// Mitsubishi GX Works2 project: PLC_GROUP_22   PLC: FX3G

// global labels: Global1
VAR_GLOBAL
  StartDayButton AT X007 : BOOL;  (* Switching it starts the work day *)
  ActiveDayLamp AT Y007 : BOOL;  (* A light that is on as long as the work day isn't over *)
  RaspberryRegister AT D1100 : REAL;  (* Raspberry inventory tracker *)
  LemonRegister AT D1102 : REAL;  (* Lemon inventory tracker *)
  PreservativeRegister AT D1104 : REAL;  (* Preservative inventory tracker *)
  GummyRegister AT D1106 : REAL;  (* Gummy inventory tracker *)
  SpecialToggle AT M0 : BOOL;  (* When Toggled - use special recpie values *)
  AnalogInput1 AT D8280 : INT;  (* Inputs a number between 1 to 10 to determine which type of popsicle to manufacture *)
  SaveAnalogInput AT D1108 : REAL;  (* Saves the value of toggled input, connects to a Onctroller to determine M0 *)
  EmergencySwitch AT X005 : BOOL;  (* Emergency break *)
  EmergencyFlag AT M2 : BOOL;  (* Signals to break the program *)
  RasperrySpecialRequirement AT E385.0 : REAL;  (* Raspberry Special requirement *)
  PreservativeSpecialRequirement AT E210.0 : REAL;  (* Preservative special recipe requirement *)
  GummySpecialRequirement AT E70.0 : REAL;  (* Gummy special recipe requirement *)
  RasperryRequirement AT E280.0 : REAL;  (* Rasperry regular recipe requirement *)
  LemonRequirement AT E455.0 : REAL;  (* Lemon regular recipe Requirement *)
  PreservativeRequirement AT E105.0 : REAL;  (* Preservative regular recipe requirement *)
  GummyRequirement AT E28.0 : REAL;  (* Gummy regular recipe requirement *)
  IceCreamStartSwitch AT X001 : BOOL;  (* When toggled - start making ice cream *)
  IceCreamMakingTimer AT TC0 : BOOL;  (* Signals if the ice cream making timer finished *)
  Constant50 AT K050 : INT;  (* The it takes to mix the ice cream *)
  IceCreamLamp AT Y000 : BOOL;  (* Signals Ice cream making in process *)
  IceCreamCompletionTimer AT TS0 : BOOL;  (* Signals the system ice cream completion *)
  CoolingSwitch AT X002 : BOOL;  (* Switch starting the cooling process *)
  IceCreamCompletionFlag AT M4 : BOOL;  (* Signals the system's ice cream completion *)
  CoolingFinishFlag AT M5 : BOOL;  (* Flag signaling the ice cream cooling ended *)
  MixingContainer AT D1110 : REAL;  (* The tank where ice cream and gummy are mixed in *)
  MixTimer AT TC1 : BOOL;  (* The time to mix special ice cream *)
  SpecialMixDuration AT K050 : INT;  (* Ice cream making time *)
  MixFinishFlag AT M7 : BOOL;  (* Signals end of mixing process *)
  RegularMixDuration AT K030 : INT;  (* The time it takes to mix regular ice cream *)
  FirstBlinkTimer AT TC3 : BOOL;  (* Timer for the first blinking lamp *)
  FirstBlinkDuration AT K005 : INT;  (* Lasts for half a second *)
  SecondBlinkTimer AT TC4 : BOOL;  (* Timer for the second blinking lamp *)
  SecondBlinkDuration AT K005 : INT;  (* Lasts for half a second *)
  FirstBlinkCompletion AT TS3 : BOOL;  (* Siignals that the first blink ended *)
  SecondBlinkCompletion AT TS4 : BOOL;  (* Signals that the first blink ended *)
  FirstBlinkLight AT Y005 : BOOL;  (* The first light that blinks during mixing *)
  SecondBlinkLight AT Y006 : BOOL;  (* The second light that blinks during mixing *)
  MixTimerFlag AT TS1 : BOOL;  (* Signals if the mixing time ended *)
  TotalPackages AT D1112 : REAL;  (* The amount of packed boxes of 7 popsicles each *)
END_VAR
VAR_GLOBAL CONSTANT
  OneMorePackage : REAL := 1.0;  (* The num ber 1, for adding 1 to the finished packages register *)
END_VAR
VAR_GLOBAL
  RasperryIceCreamContainer AT D1114 : REAL;  (* Simulates Rasp. IceCream Container *)
  LemonIceCreamContainer AT D1116 : REAL;  (* Simulates Lemon IceCream Container *)
  LemonSpecialRequirement AT E665.0 : REAL;  (* Lemon special recipe requirement *)
  RasperryIceCreamSpecialRecepie AT E560.0 : REAL;  (* The amount of rasperry Icecream produced in 1 special production run *)
  LemonIceCreamSpecialRecepie AT E700.0 : REAL;  (* The amount of lemon icecream for 1 special production run *)
  RasperryIceCreamRegularRecepie AT E350.0 : REAL;  (* The amount of raspberry Icecream produced in 1 regular production run *)
  LemonIceCreamRegularRecepie AT E490.0 : REAL;  (* The amount of lemon ice cream for 1 regular production run *)
  RasperryCoolingContainer AT D1118 : REAL;  (* Simulates Rasperry cooling container *)
  LemonCoolingCOntainer AT D1120 : REAL;  (* Simulates Lemon cooling container *)
  CoolingStart AT M9 : BOOL;  (* Signals the cooling process has begun *)
  CoolingTimer AT TC5 : BOOL;  (* Timer for the cooling process *)
  CoolingTimerConstant AT K80 : INT;  (* Duration of the cooling process *)
  CoolingTImerSignal AT TS5 : BOOL;  (* Signals the cooling process has ended *)
  TempratureSensor AT X003 : BOOL;  (* TempratureSensor *)
  CoolingLamp AT Y002 : BOOL;  (* Cooling Process Lamp *)
  TempreatureSensorFlag AT M10 : BOOL;  (* Signals the temeprature sensor is on *)
  BlinkHelperFlag AT M11 : BOOL;  (* A helper variable for the blinking process *)
  MixTimerRegular AT TC2 : BOOL;  (* The time to mix regular ice cream *)
  MixTimerRegularFlag AT TS2 : BOOL;  (* The time to mix special ice cream *)
  TenFloat AT E10.0 : REAL;  (* The number 10 *)
  RaspberryINIT AT D1222 : REAL;  (* The initial value the inventory recieves at start of day *)
  LemonINIT AT D1224 : REAL;  (* The initial value the inventory recieves at start of day *)
  PerservartiveINIT AT D1226 : REAL;  (* The initial value the inventory recieves at start of day *)
  GummyINIT AT D1228 : REAL;  (* The initial value the inventory recieves at start of day *)
  Zero AT K0 : INT;  (* The number zero, used to reset variables *)
  ResetRegisterSize AT K101 : INT;  (* The range of data registers to reset *)
  FloatConstant5 AT E5.0 : REAL;  (* The maximum input for regular recipe *)
  FloatConstant6 AT E6.0 : REAL;  (* The minimum input for special recipe *)
  FloatConstant10 AT E10.0 : REAL;  (* The maximum input for our program *)
  Float400 AT E400.0 : REAL;  (* Float 400 *)
  GreaterThan5 AT M12 : BOOL;  (* Flag signaling input is greater than 5 *)
  GreaterEqual6Flag AT M13 : BOOL;  (* Flag signaling input is greater equal than 5 *)
  GreaterThan10 AT M14 : BOOL;  (* flag signifies input is greater than 10 *)
  InputEmergencyFlag AT M15 : BOOL;  (* Flag signifies the input is invalid and should crash *)
  Float40 AT E40.0 : REAL;  (* Float 40 *)
  AnalogOutput AT D8282 : INT;  (* Analog output register *)
  LowRasperryFlag AT M16 : BOOL;
  LowLemonFlag AT M17 : BOOL;
  LowPerservativeFlag AT M18 : BOOL;
  LowGummyFlag AT M19 : BOOL;
  Y7Flag AT M20 : BOOL;
  Y0Flag AT M21 : BOOL;
  Y2Flag AT M22 : BOOL;
  ResetFlag AT M23 : BOOL;
END_VAR

// task Task_01 (event TRUE, interval 0, priority 31): POU_01

PROGRAM POU_01
(* structured ladder/FBD written out as ST: instructions are called as NAME(EN, inputs, outputs); _pN, _eN, _tN stand for wires *)
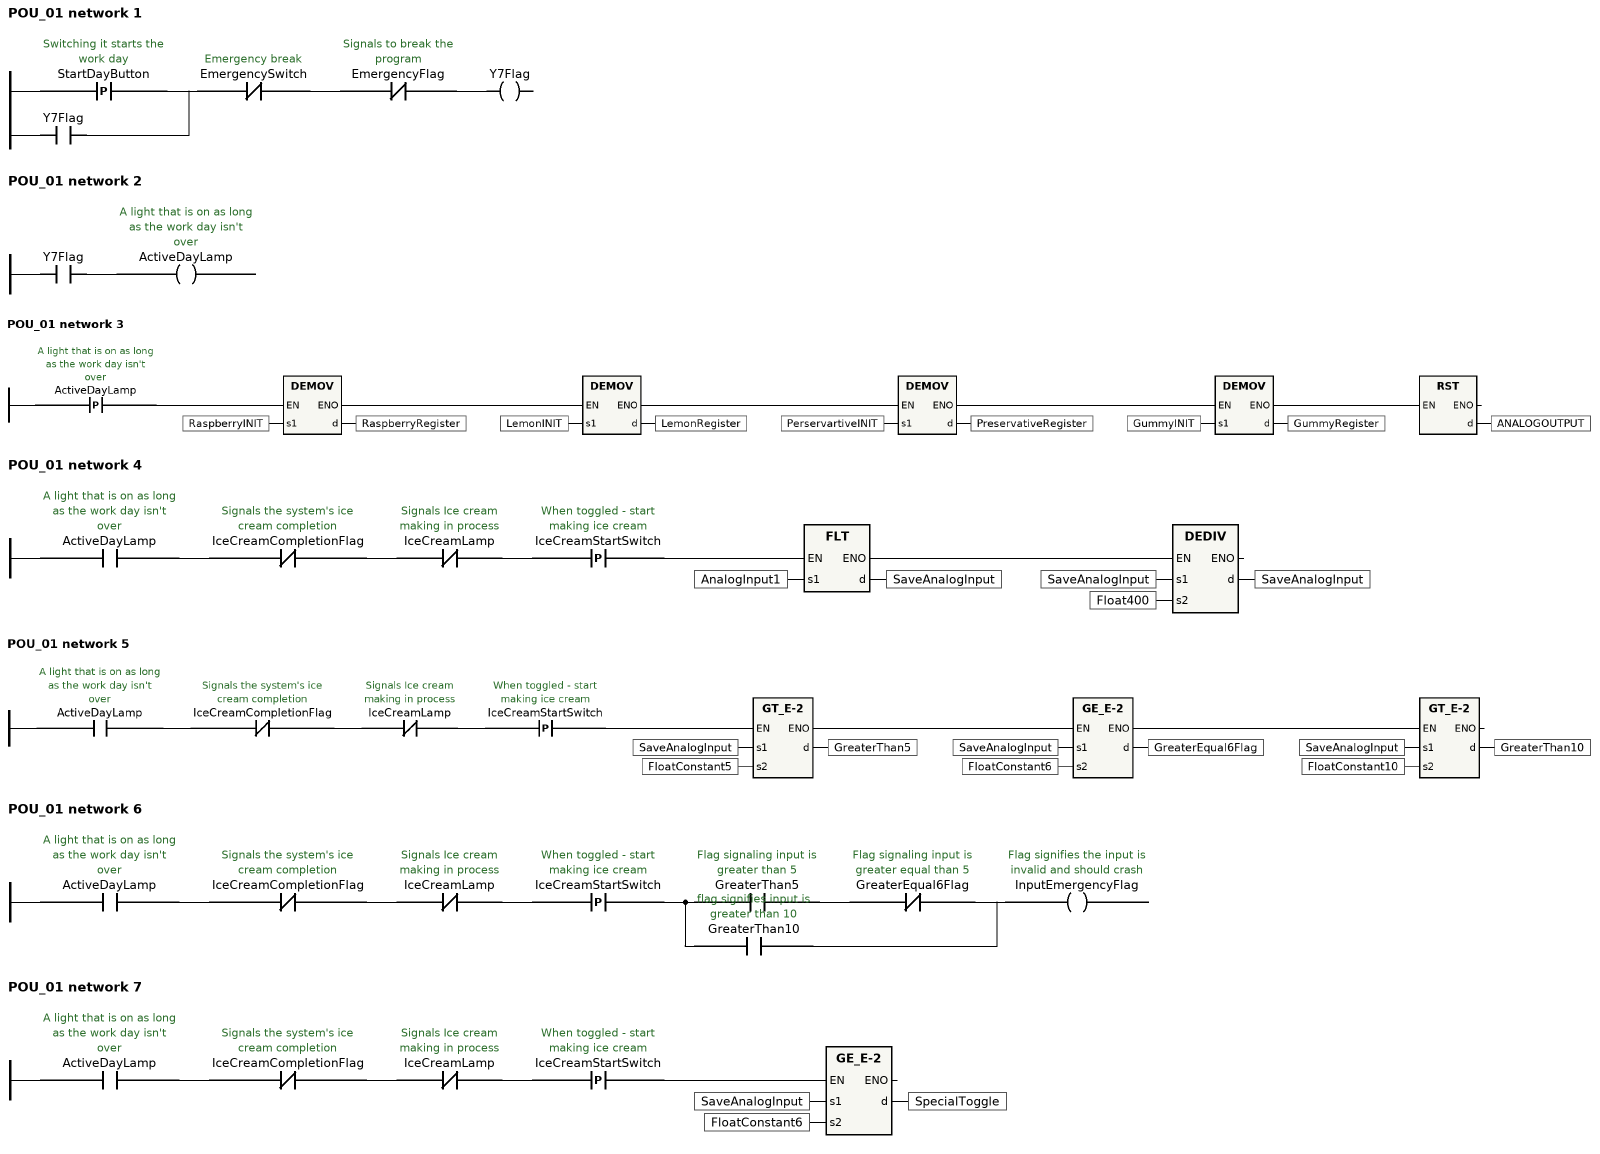
(* network 1 Start the work day *)
Y7Flag := ((LDP(TRUE, StartDayButton) OR Y7Flag) AND NOT EmergencySwitch) AND NOT EmergencyFlag;
(* network 2 Turn 7 lamp on *)
ActiveDayLamp := Y7Flag;
(* network 3 Recieve INIT vals *)
_e1 := DEMOV(LDP(TRUE, ActiveDayLamp), RaspberryINIT, RaspberryRegister);
_e2 := DEMOV(_e1, LemonINIT, LemonRegister);
_e3 := DEMOV(_e2, PerservartiveINIT, PreservativeRegister);
_e4 := DEMOV(_e3, GummyINIT, GummyRegister);
RST(_e4, ANALOGOUTPUT);
(* network 4 Transform input *)
_e1 := FLT(ActiveDayLamp AND NOT IceCreamCompletionFlag AND NOT IceCreamLamp AND LDP(TRUE, IceCreamStartSwitch), AnalogInput1, SaveAnalogInput);
DEDIV(_e1, SaveAnalogInput, Float400, SaveAnalogInput);
(* network 5 Input range flags *)
_e1 := GT_E(ActiveDayLamp AND NOT IceCreamCompletionFlag AND NOT IceCreamLamp AND LDP(TRUE, IceCreamStartSwitch), SaveAnalogInput, FloatConstant5, GreaterThan5);
_e2 := GE_E(_e1, SaveAnalogInput, FloatConstant6, GreaterEqual6Flag);
GT_E(_e2, SaveAnalogInput, FloatConstant10, GreaterThan10);
(* network 6 Input validation *)
_p1 := ActiveDayLamp AND NOT IceCreamCompletionFlag AND NOT IceCreamLamp AND LDP(TRUE, IceCreamStartSwitch);
InputEmergencyFlag := (_p1 AND GreaterThan5 AND NOT GreaterEqual6Flag) OR (_p1 AND GreaterThan10);
(* network 7 Special check *)
GE_E(ActiveDayLamp AND NOT IceCreamCompletionFlag AND NOT IceCreamLamp AND LDP(TRUE, IceCreamStartSwitch), SaveAnalogInput, FloatConstant6, SpecialToggle);
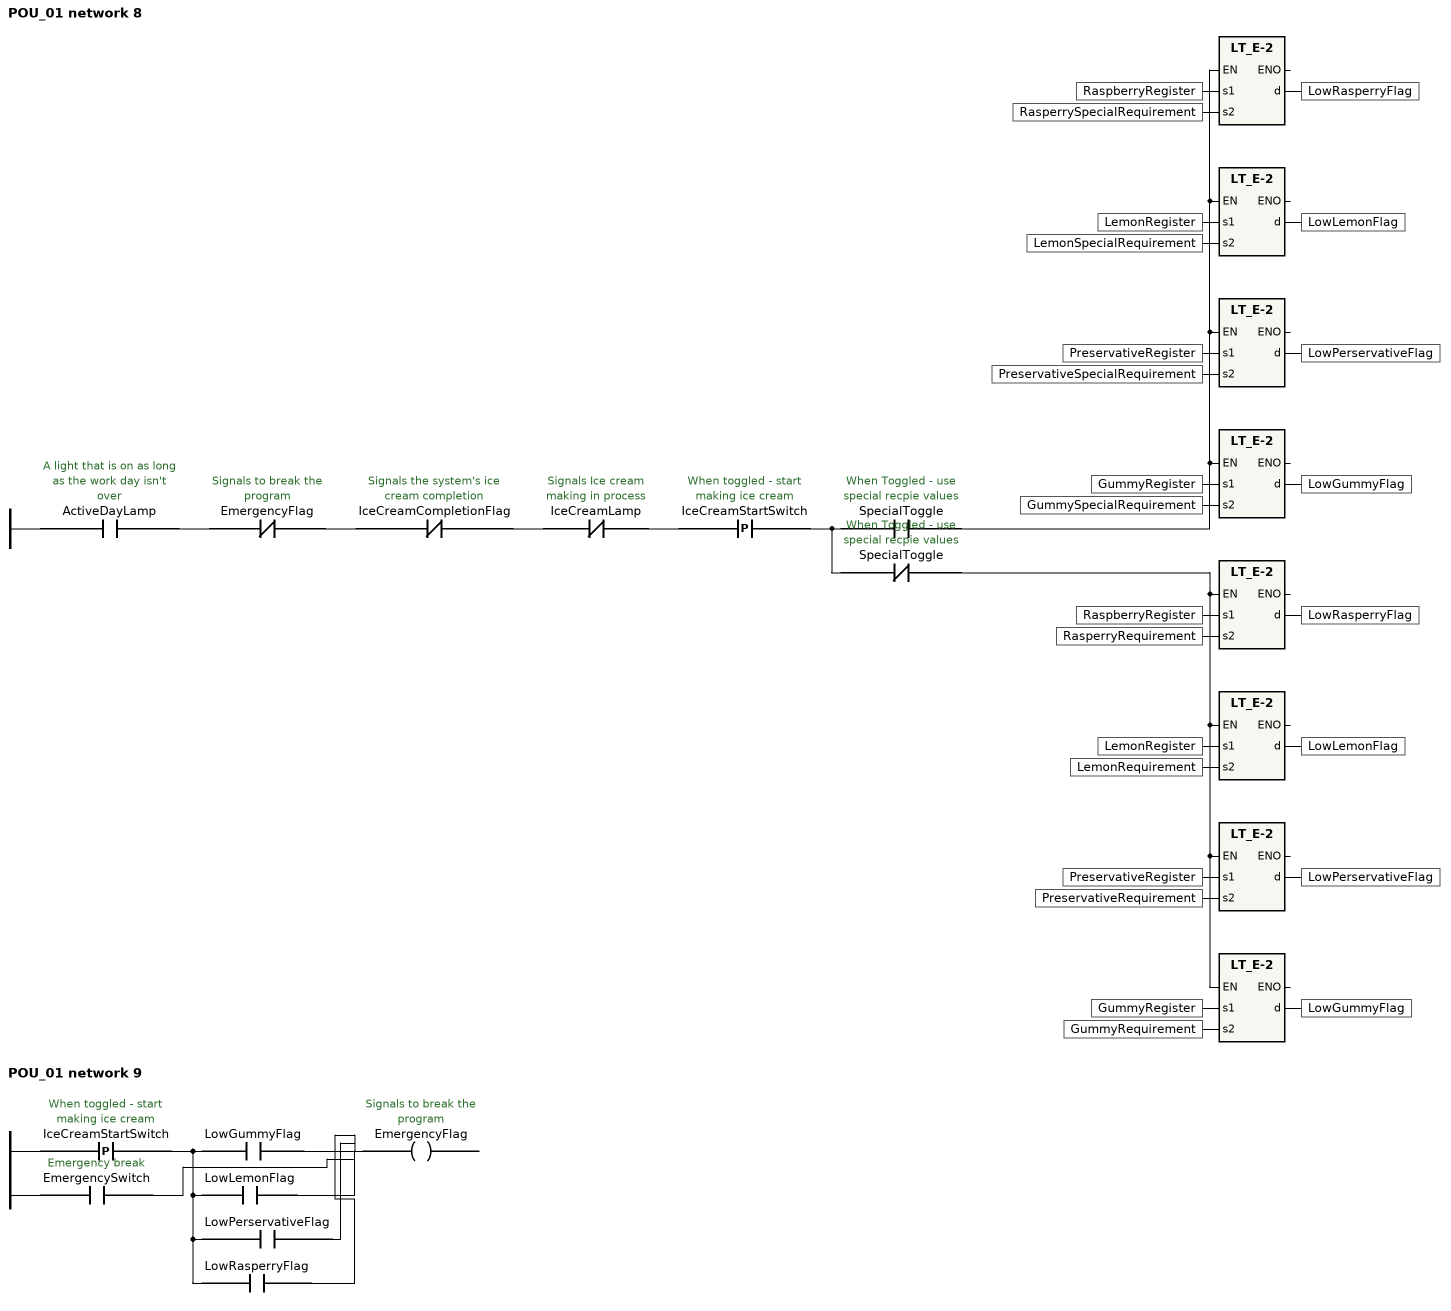
(* network 8 Inventory check *)
_p1 := ActiveDayLamp AND NOT EmergencyFlag AND NOT IceCreamCompletionFlag AND NOT IceCreamLamp AND LDP(TRUE, IceCreamStartSwitch);
_p2 := _p1 AND SpecialToggle;
LT_E(_p2, RaspberryRegister, RasperrySpecialRequirement, LowRasperryFlag);
LT_E(_p2, LemonRegister, LemonSpecialRequirement, LowLemonFlag);
LT_E(_p2, PreservativeRegister, PreservativeSpecialRequirement, LowPerservativeFlag);
LT_E(_p2, GummyRegister, GummySpecialRequirement, LowGummyFlag);
_p3 := _p1 AND NOT SpecialToggle;
LT_E(_p3, RaspberryRegister, RasperryRequirement, LowRasperryFlag);
LT_E(_p3, LemonRegister, LemonRequirement, LowLemonFlag);
LT_E(_p3, PreservativeRegister, PreservativeRequirement, LowPerservativeFlag);
LT_E(_p3, GummyRegister, GummyRequirement, LowGummyFlag);
(* network 9 Inventory check flag *)
_p1 := LDP(TRUE, IceCreamStartSwitch);
EmergencyFlag := (_p1 AND LowGummyFlag) OR (_p1 AND LowLemonFlag) OR (_p1 AND LowPerservativeFlag) OR (_p1 AND LowRasperryFlag) OR EmergencySwitch;
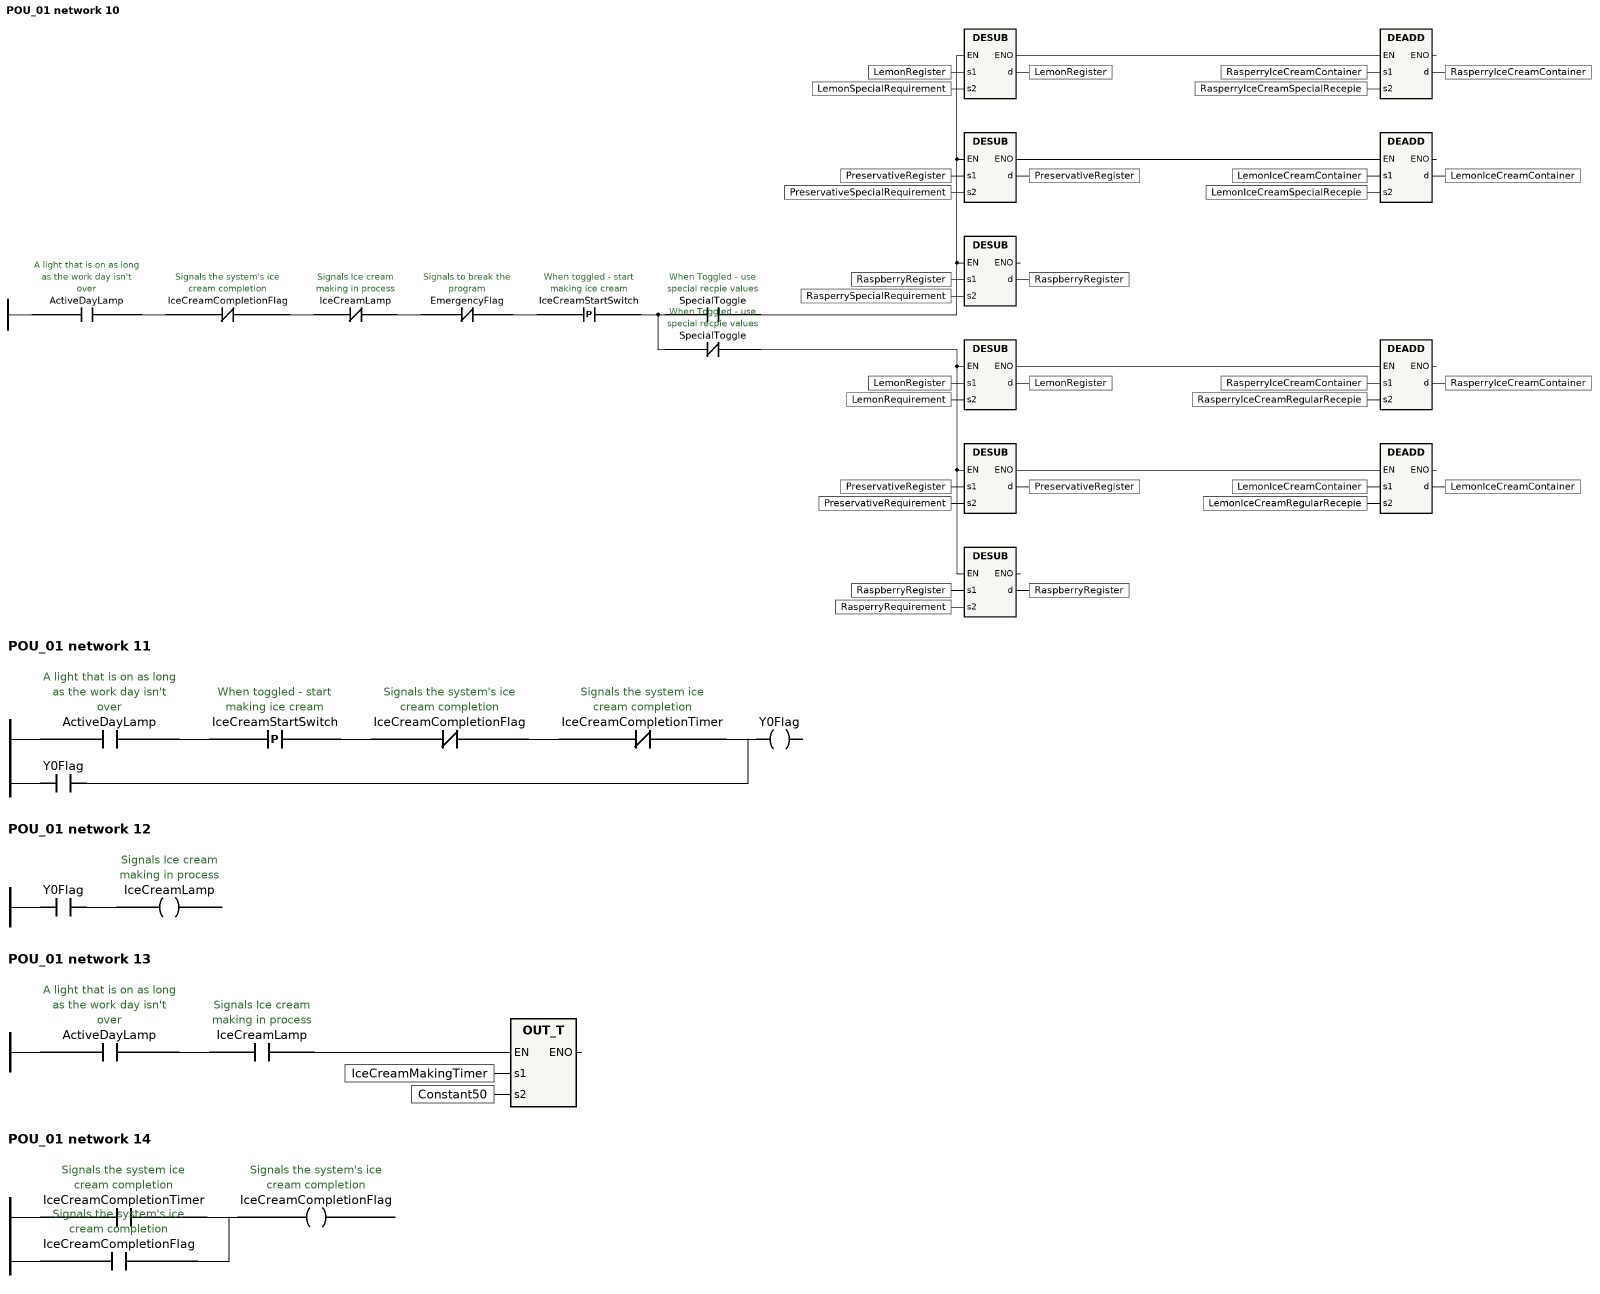
(* network 10 Transfer to Containe *)
_p1 := ActiveDayLamp AND NOT IceCreamCompletionFlag AND NOT IceCreamLamp AND NOT EmergencyFlag AND LDP(TRUE, IceCreamStartSwitch);
_p2 := _p1 AND SpecialToggle;
_e3 := DESUB(_p2, LemonRegister, LemonSpecialRequirement, LemonRegister);
DEADD(_e3, RasperryIceCreamContainer, RasperryIceCreamSpecialRecepie, RasperryIceCreamContainer);
_e4 := DESUB(_p2, PreservativeRegister, PreservativeSpecialRequirement, PreservativeRegister);
DEADD(_e4, LemonIceCreamContainer, LemonIceCreamSpecialRecepie, LemonIceCreamContainer);
DESUB(_p2, RaspberryRegister, RasperrySpecialRequirement, RaspberryRegister);
_p5 := _p1 AND NOT SpecialToggle;
_e6 := DESUB(_p5, LemonRegister, LemonRequirement, LemonRegister);
DEADD(_e6, RasperryIceCreamContainer, RasperryIceCreamRegularRecepie, RasperryIceCreamContainer);
_e7 := DESUB(_p5, PreservativeRegister, PreservativeRequirement, PreservativeRegister);
DEADD(_e7, LemonIceCreamContainer, LemonIceCreamRegularRecepie, LemonIceCreamContainer);
DESUB(_p5, RaspberryRegister, RasperryRequirement, RaspberryRegister);
(* network 11 IceCreamLamp flag *)
Y0Flag := (ActiveDayLamp AND LDP(TRUE, IceCreamStartSwitch) AND NOT IceCreamCompletionFlag AND NOT IceCreamCompletionTimer) OR Y0Flag;
(* network 12 IceCreamLamp on *)
IceCreamLamp := Y0Flag;
(* network 13 IceCreamMaking Timer *)
OUT_T(ActiveDayLamp AND IceCreamLamp, IceCreamMakingTimer, Constant50);
(* network 14 Turn on icecreamflag *)
IceCreamCompletionFlag := IceCreamCompletionTimer OR IceCreamCompletionFlag;
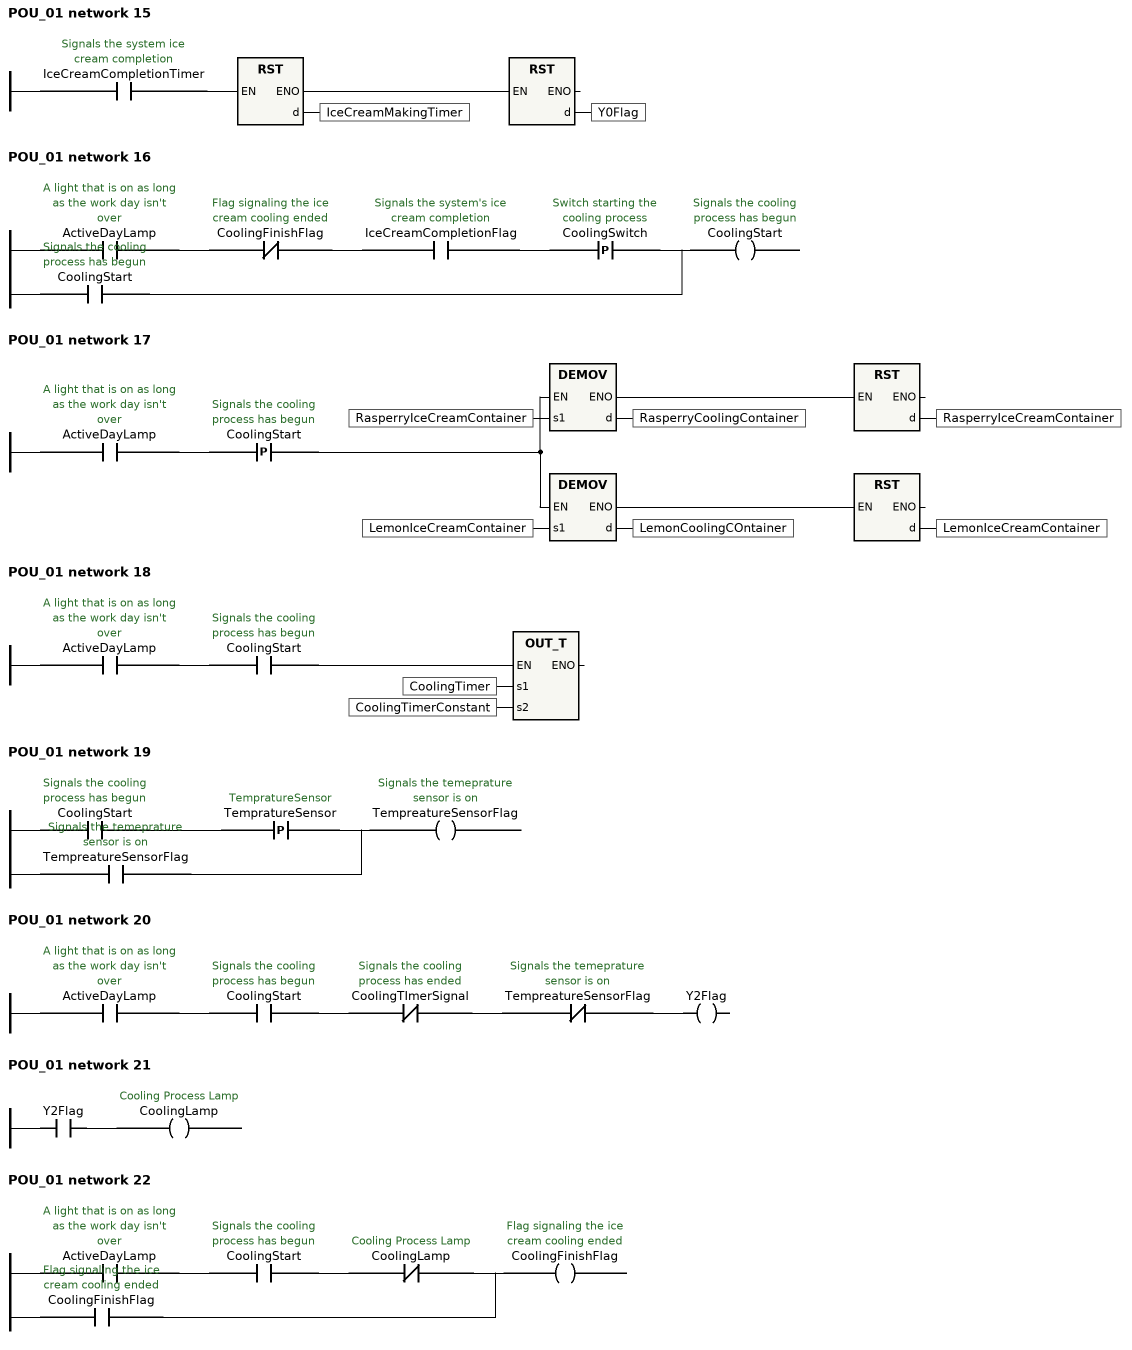
(* network 15 Reset local variable *)
_e1 := RST(IceCreamCompletionTimer, IceCreamMakingTimer);
RST(_e1, Y0Flag);
(* network 16 Start cooling *)
CoolingStart := (ActiveDayLamp AND NOT CoolingFinishFlag AND IceCreamCompletionFlag AND LDP(TRUE, CoolingSwitch)) OR CoolingStart;
(* network 17 Transfer to cool *)
_p1 := ActiveDayLamp AND LDP(TRUE, CoolingStart);
_e2 := DEMOV(_p1, RasperryIceCreamContainer, RasperryCoolingContainer);
RST(_e2, RasperryIceCreamContainer);
_e3 := DEMOV(_p1, LemonIceCreamContainer, LemonCoolingCOntainer);
RST(_e3, LemonIceCreamContainer);
(* network 18 Start Cooling Timer *)
OUT_T(ActiveDayLamp AND CoolingStart, CoolingTimer, CoolingTimerConstant);
(* network 19 Signal 10C Sensor *)
TempreatureSensorFlag := (CoolingStart AND LDP(TRUE, TempratureSensor)) OR TempreatureSensorFlag;
(* network 20 Lamp on conditions *)
Y2Flag := ActiveDayLamp AND CoolingStart AND NOT CoolingTImerSignal AND NOT TempreatureSensorFlag;
(* network 21 flag to lamp conn *)
CoolingLamp := Y2Flag;
(* network 22 Flag cooling finish *)
CoolingFinishFlag := (ActiveDayLamp AND CoolingStart AND NOT CoolingLamp) OR CoolingFinishFlag;
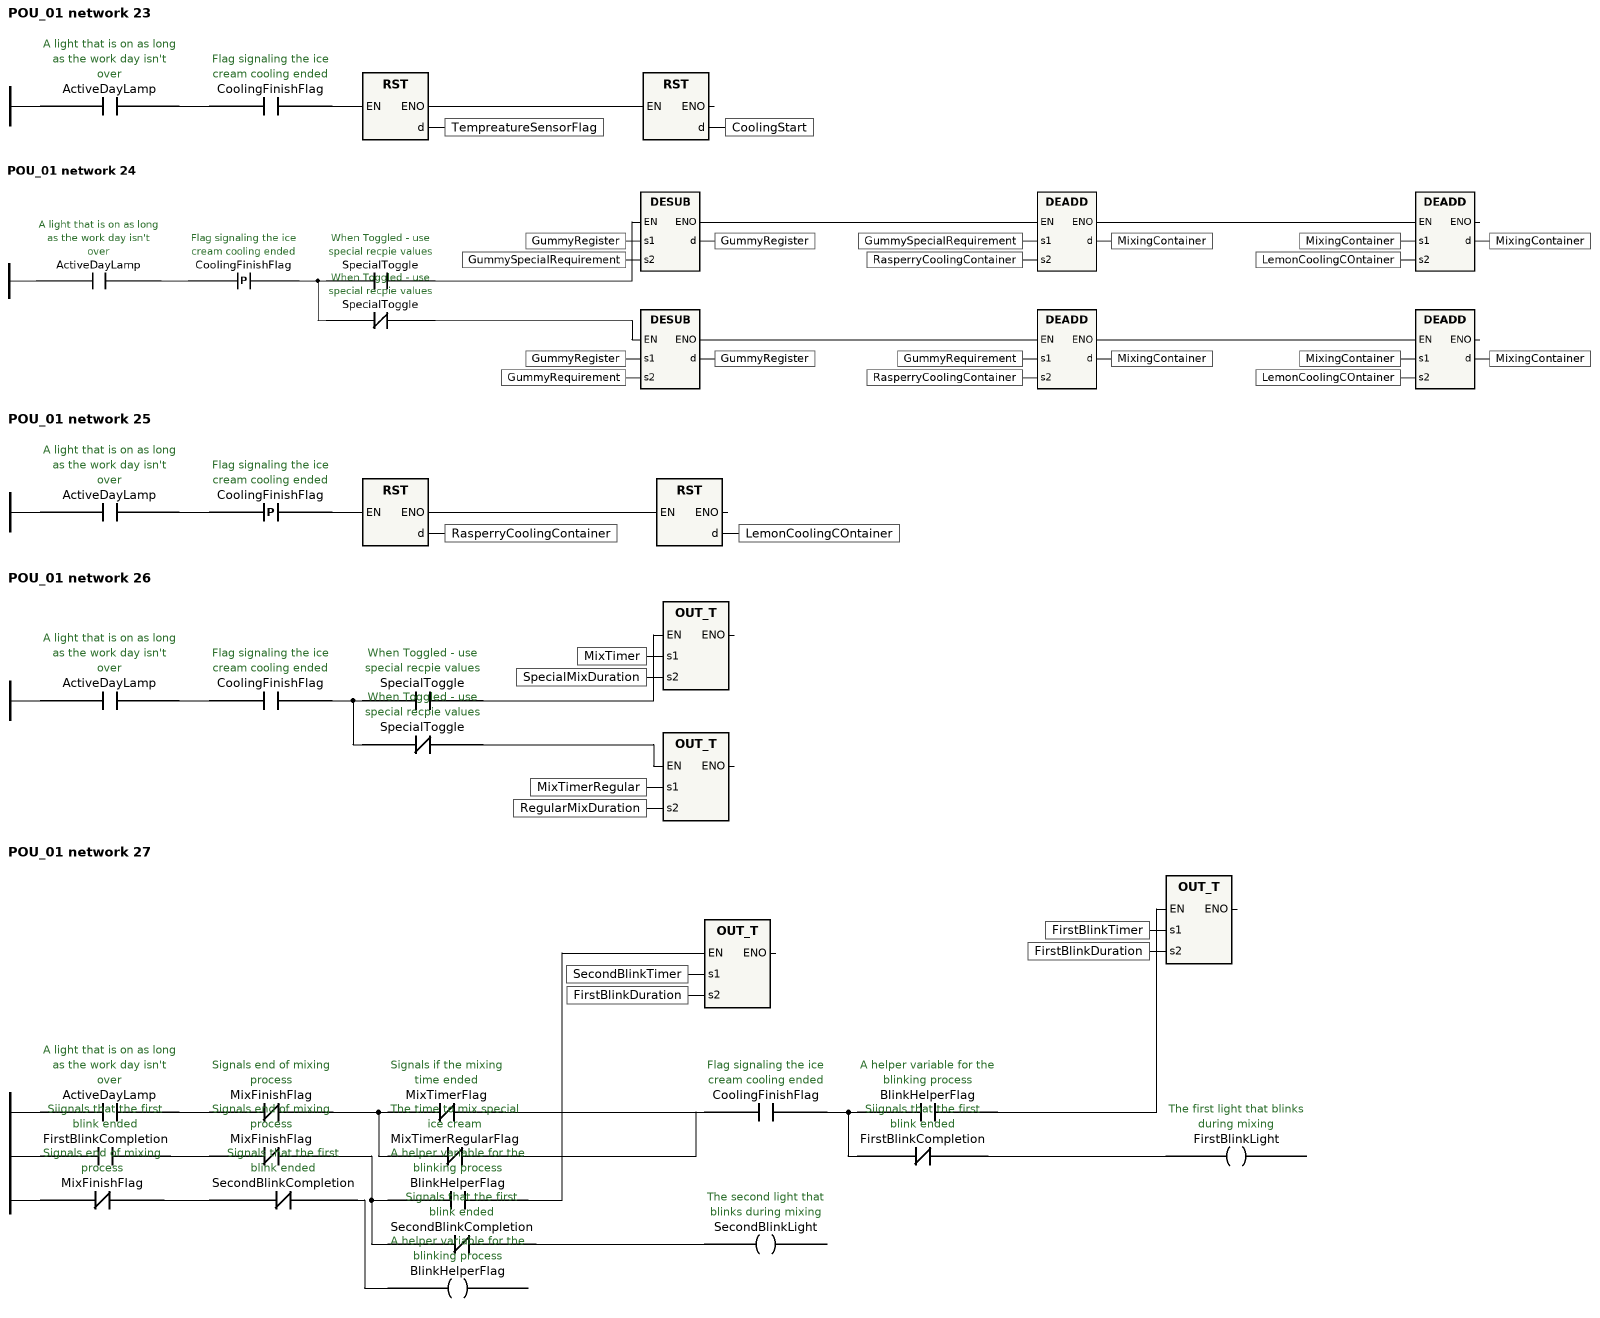
(* network 23 Reset vars *)
_e1 := RST(ActiveDayLamp AND CoolingFinishFlag, TempreatureSensorFlag);
RST(_e1, CoolingStart);
(* network 24 Add to mixing tank *)
_p1 := ActiveDayLamp AND LDP(TRUE, CoolingFinishFlag);
_e2 := DESUB(_p1 AND SpecialToggle, GummyRegister, GummySpecialRequirement, GummyRegister);
_e3 := DEADD(_e2, GummySpecialRequirement, RasperryCoolingContainer, MixingContainer);
DEADD(_e3, MixingContainer, LemonCoolingCOntainer, MixingContainer);
_e4 := DESUB(_p1 AND NOT SpecialToggle, GummyRegister, GummyRequirement, GummyRegister);
_e5 := DEADD(_e4, GummyRequirement, RasperryCoolingContainer, MixingContainer);
DEADD(_e5, MixingContainer, LemonCoolingCOntainer, MixingContainer);
(* network 25 Zero cooling cont *)
_e1 := RST(ActiveDayLamp AND LDP(TRUE, CoolingFinishFlag), RasperryCoolingContainer);
RST(_e1, LemonCoolingCOntainer);
(* network 26 Setting mixing timer *)
_p1 := ActiveDayLamp AND CoolingFinishFlag;
OUT_T(_p1 AND SpecialToggle, MixTimer, SpecialMixDuration);
OUT_T(_p1 AND NOT SpecialToggle, MixTimerRegular, RegularMixDuration);
(* network 27 1st blink check *)
_p1 := ActiveDayLamp AND NOT MixFinishFlag;
_p2 := ((_p1 AND NOT MixTimerFlag) OR (_p1 AND NOT MixTimerRegularFlag)) AND CoolingFinishFlag;
OUT_T(_p2 AND BlinkHelperFlag, FirstBlinkTimer, FirstBlinkDuration);
FirstBlinkLight := _p2 AND NOT FirstBlinkCompletion;
_p3 := FirstBlinkCompletion AND NOT MixFinishFlag;
OUT_T(_p3 AND BlinkHelperFlag, SecondBlinkTimer, FirstBlinkDuration);
SecondBlinkLight := _p3 AND NOT SecondBlinkCompletion;
BlinkHelperFlag := NOT MixFinishFlag AND NOT SecondBlinkCompletion;
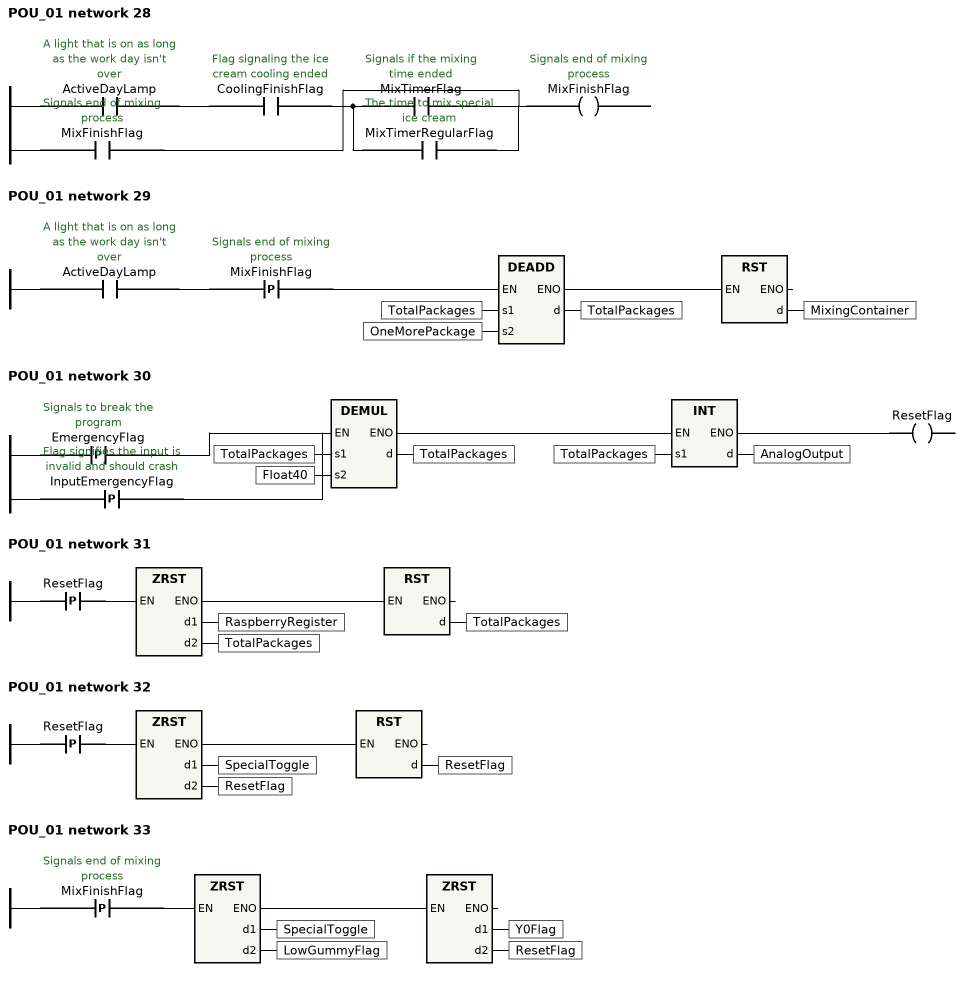
(* network 28 Flag mix completion *)
_p1 := ActiveDayLamp AND CoolingFinishFlag;
MixFinishFlag := (_p1 AND MixTimerFlag) OR (_p1 AND MixTimerRegularFlag) OR MixFinishFlag;
(* network 29 add to package count *)
_e1 := DEADD(ActiveDayLamp AND LDP(TRUE, MixFinishFlag), TotalPackages, OneMorePackage, TotalPackages);
RST(_e1, MixingContainer);
(* network 30 calculate packages *)
_e1 := DEMUL(LDP(TRUE, EmergencyFlag) OR LDP(TRUE, InputEmergencyFlag), TotalPackages, Float40, TotalPackages);
_e2 := INT(_e1, TotalPackages, AnalogOutput);
ResetFlag := _e2;
(* network 31 Emergeny Reset block *)
_e1 := ZRST(LDP(TRUE, ResetFlag), RaspberryRegister, TotalPackages);
RST(_e1, TotalPackages);
(* network 32 *)
_e1 := ZRST(LDP(TRUE, ResetFlag), SpecialToggle, ResetFlag);
RST(_e1, ResetFlag);
(* network 33 Emergeny Reset block *)
_e1 := ZRST(LDP(TRUE, MixFinishFlag), SpecialToggle, LowGummyFlag);
ZRST(_e1, Y0Flag, ResetFlag);
END_PROGRAM
